// TIA Portal V15.1 export
// export: Created 2026-01-09T13:45:14.0134605Z, ExportSetting WithDefaults, WithReadOnly, DisplayName Totally Integrated Automation Portal, DisplayVersion V15.1 Update 8, DisplayName TIA Portal Openness, DisplayVersion V15.1 Update 8, DisplayName STEP 7 Professional, DisplayVersion V15.1 Update 8, DisplayName WinCC Advanced, DisplayVersion V15.1 Update 8
FUNCTION_BLOCK "5.ADDITIVES_PULE"   // FB5, LAD
{ S7_Optimized_Access := 'TRUE' }
VERSION : 0.1
// stored: AutoNumber false, CodeModifiedDate 2024-07-29T16:22:18.8856203Z, CompileDate 2025-08-30T17:40:35.1271729Z, CreationDate 2024-10-12T12:36:08.0193576Z, DownloadWithoutReinit false, HandleErrorsWithinBlock false, InterfaceModifiedDate 2024-07-29T16:20:48.5427985Z, IsConsistent true, IsIECCheckEnabled false, IsKnowHowProtected false, IsRetainMemResEnabled false, IsWriteProtected false, LibraryConformanceStatus The object is library-conformant., MemoryReserve 100, ModifiedDate 2024-07-29T16:22:18.8856203Z, ParameterModified 2024-07-29T16:20:48.5427985Z, PLCSimAdvancedSupport false, SetENOAutomatically False, StructureModified 2024-07-29T16:20:48.5427985Z, UDAEnableTagReadback false
   VAR_INPUT
      "Xung In" : DWord;
      Reset : Bool;
      "Set Tai" : Bool;
      "Khoi Luong Calib" : Real;
   END_VAR
   VAR_OUTPUT
      "Khoi Luong Out" : Real;
      "Xung Out" : Real;
   END_VAR
   VAR RETAIN
      "Xu In" : Real;
      "He So" : Real;
      "Xu Calib" : Real;
      "Kl Calib" : Real;
   END_VAR
   VAR
      M1 : Bool;
   END_VAR
   VAR_TEMP
      Conv : DInt;
   END_VAR
BEGIN

REGION Network 1
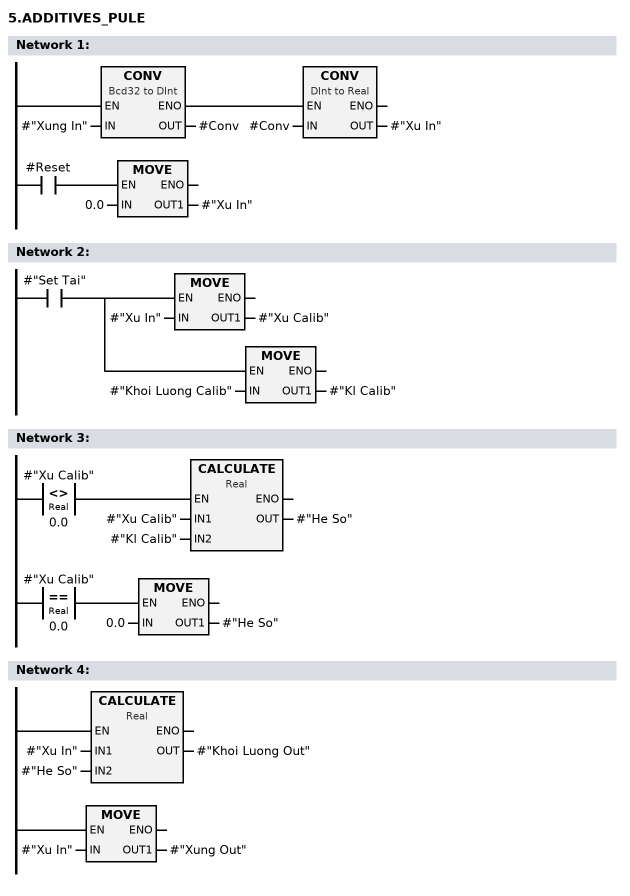
   RUNG wire#powerrail
      { S7_Templates := "[SrcType := Bcd32, DestType := DInt]" } Convert(in := #"Xung In", out => #Conv)
      { S7_Templates := "[SrcType := DInt, DestType := Real]" } Convert(in := #Conv, out => #"Xu In")
   END_RUNG
   RUNG wire#powerrail
      Contact( #Reset )
      Move(in := 0.0, out1 => #"Xu In")
   END_RUNG
   // the same network as SCL:
   #Conv := BCD32_TO_DINT(#"Xung In");
   #"Xu In" := DINT_TO_REAL(#Conv);
   IF #Reset THEN #"Xu In" := 0.0; END_IF;
END_REGION

REGION Network 2
   RUNG wire#powerrail
      Contact( #"Set Tai" )
      wire#w1
      Move(in := #"Xu In", out1 => #"Xu Calib")
   END_RUNG
   RUNG wire#w1
      Move(in := #"Khoi Luong Calib", out1 => #"Kl Calib")
   END_RUNG
   // the same network as SCL:
   IF #"Set Tai" THEN
       #"Xu Calib" := #"Xu In";
       #"Kl Calib" := #"Khoi Luong Calib";
   END_IF;
END_REGION

REGION Network 3
   RUNG wire#powerrail
      { S7_Templates := "SrcType := Real" } NE_Contact(in1 := #"Xu Calib", in2 := 0.0)
      { S7_Templates := "SrcType := Real"; S7_Expression := "IN2/IN1" } Calculate(in1 := #"Xu Calib", in2 := #"Kl Calib", out => #"He So")
   END_RUNG
   RUNG wire#powerrail
      { S7_Templates := "SrcType := Real" } EQ_Contact(in1 := #"Xu Calib", in2 := 0.0)
      Move(in := 0.0, out1 => #"He So")
   END_RUNG
   // the same network as SCL:
   IF #"Xu Calib" <> 0.0 THEN #"He So" := #"Kl Calib"/#"Xu Calib"; END_IF;
   IF #"Xu Calib" = 0.0 THEN #"He So" := 0.0; END_IF;
END_REGION

REGION Network 4
   RUNG wire#powerrail
      { S7_Templates := "SrcType := Real"; S7_Expression := "IN1*IN2" } Calculate(in1 := #"Xu In", in2 := #"He So", out => #"Khoi Luong Out")
   END_RUNG
   RUNG wire#powerrail
      Move(in := #"Xu In", out1 => #"Xung Out")
   END_RUNG
   // the same network as SCL:
   #"Khoi Luong Out" := #"Xu In"*#"He So";
   #"Xung Out" := #"Xu In";
END_REGION
END_FUNCTION_BLOCK
